{attribute 'qualified_only'}
VAR_GLOBAL
	sNetId: T_AmsNetId := '5.53.143.24.1.1';
	nPort: T_AmsPort := 851;	
END_VAR

(* stored: Version 1.1.0.1, ProductVersion 3.1.4024.11
   GVL ReactorAms: Id {5f549537-136b-42af-966f-98c78cd25f00} *)
